TYPE "ST_SpkCylHal"
VERSION : 0.1
   STRUCT
      Extend : Bool;               // valve coils (outputs)
      Retract : Bool;
      Extended : Bool;             // end-position sensors (inputs)
      Retracted : Bool;
   END_STRUCT;

END_TYPE
